Staubli VAL3: lists_num.pjx

Parameters version=s8.13.1Cs9_BS2800 stackSize=5000 millimeterUnit=true
Program file=start.pgx
Program file=stop.pgx
Data file=lists_num.dtx
